PROGRAM MAIN
VAR
END_VAR

END_PROGRAM

(* stored: Version 1.1.0.1
   POU MAIN: Id {f6b5c2c0-bb0f-4a89-8be5-3f2e29d89415} *)
